Fanuc KAREL source: ka00078.KL

PROGRAM KA00078
%NOLOCKGROUP
VAR
SRC : XYZWPREXT;DST : XYZWPR
BEGIN
--
SRC.X=1.0
DST=SRC
END KA00078
